// TIA Portal project "TranMinhQuan_19151078" (V15)

(* hardware
DEVICE "S7-1200 station_1"  S7-1200 Station
   slot 0: "Rack_0"  S7-1200 Rack  Rack  V1.0
   slot 1: "PLC_1"  CPU 1214C DC/DC/DC  6ES7 214-1AG40-0XB0  V4.2
*)

// ===== PLC "PLC_1"  CPU 1214C DC/DC/DC =====

VAR_GLOBAL   // PLC tag table "Default tag table"
   "FOR" AT %I0.0 : Bool;
   "LEFT" AT %Q0.1 : Bool;
   "LS1" AT %I0.2 : Bool;
   "RIGHT" AT %Q0.0 : Bool;
   "LS2" AT %I0.3 : Bool;
   "STOP" AT %I0.1 : Bool;
END_VAR

// folder: System blocks/Program resources

DATA_BLOCK "T0"   // DB1
{ S7_Optimized_Access := 'TRUE' }
AUTHOR : Simatic
FAMILY : IEC
NAME : IEC_TMR
VERSION : 1.0
// stored: InstanceOfName IEC_TIMER
"IEC_TIMER"
BEGIN
END_DATA_BLOCK

DATA_BLOCK "T1"   // DB2
{ S7_Optimized_Access := 'TRUE' }
AUTHOR : Simatic
FAMILY : IEC
NAME : IEC_TMR
VERSION : 1.0
// stored: InstanceOfName IEC_TIMER
"IEC_TIMER"
BEGIN
END_DATA_BLOCK

// folder: (top level)

ORGANIZATION_BLOCK "Main"   // OB1, LAD, ProgramCycle
TITLE = "Main Program Sweep (Cycle)"
{ S7_Optimized_Access := 'TRUE' }
VERSION : 0.1
   VAR_INPUT
      Initial_Call : Bool;   // Initial call of this OB
      Remanence : Bool;   // =True, if remanent data are available
   END_VAR
BEGIN

REGION Network 1
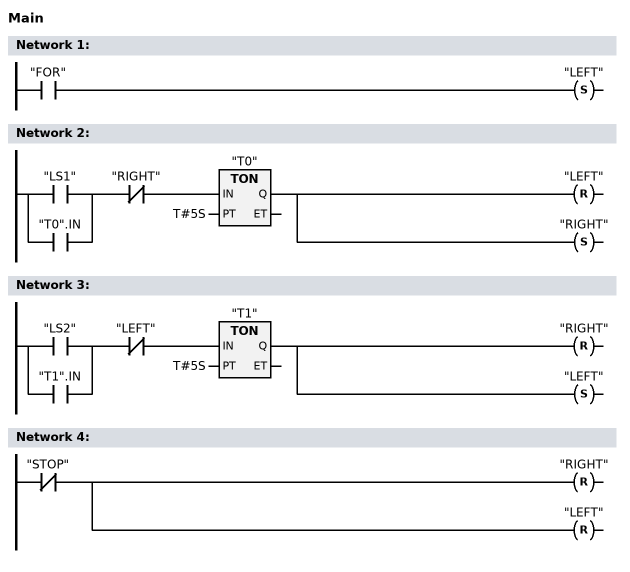
   RUNG wire#powerrail
      Contact( "FOR" )
      S_Coil( "LEFT" )
   END_RUNG
   // the same network as SCL:
   IF "FOR" THEN "LEFT" := TRUE; END_IF;
END_REGION

REGION Network 2
   "T0".TON(IN := ("LS1" OR "T0".IN) AND NOT "RIGHT", PT := T#5S);
   IF "T0".Q THEN
       "LEFT" := FALSE;
       "RIGHT" := TRUE;
   END_IF;
END_REGION

REGION Network 3
   "T1".TON(IN := ("LS2" OR "T1".IN) AND NOT "LEFT", PT := T#5S);
   IF "T1".Q THEN
       "RIGHT" := FALSE;
       "LEFT" := TRUE;
   END_IF;
END_REGION

REGION Network 4
   RUNG wire#powerrail
      I_Contact( "STOP" )
      wire#w1
      R_Coil( "RIGHT" )
   END_RUNG
   RUNG wire#w1
      R_Coil( "LEFT" )
   END_RUNG
   // the same network as SCL:
   IF NOT "STOP" THEN
       "RIGHT" := FALSE;
       "LEFT" := FALSE;
   END_IF;
END_REGION
END_ORGANIZATION_BLOCK